// TwinCAT 3 PLC project TwinCAT_NC_Sample_Flying_Saw
// libraries:
//   Tc2_Math, * (Beckhoff Automation GmbH)
//   Tc2_MC2, * (Beckhoff Automation GmbH)
//   Tc2_MC2_FlyingSaw, * (Beckhoff Automation GmbH)
//   Tc2_Standard, * (Beckhoff Automation GmbH)
//   Tc2_System, * (Beckhoff Automation GmbH)
//   Tc3_Module, * (Beckhoff Automation GmbH)
// project tree:
//   Data types/ ST_AxisIn.TcDUT, ST_Axis.TcDUT, ST_AxisOut.TcDUT
//   Global Variables/ Globale_Variablen.TcGVL, GVL_FlyingSaw.TcGVL
//   / GlobalTextList.TcGTLO, PlcTask.TcTTO, Visualization Manager.TcVMO (not stored), VISU_TASK.TcTTO
//   POUs/ FB_Motion.TcPOU, MAIN.TcPOU, PRG_FlyingSaw.TcPOU, PRG_Simulation.TcPOU
//   Visualizations/ ImagePool.TcIPO (not stored), TC_FlyingSawPage.TcVIS
// real-time tasks:
//   TASK PlcTask: cycle T#10ms, priority 20, ADS port 350
//   TASK VISU_TASK: cycle T#10ms, priority 30, ADS port 351
// motion (NC):
//   TASK NC-Task 1 SAF: cycle T#2ms, priority 4, ADS port 501
//   TASK NC-Task 1 SVB: cycle T#10ms, priority 8, ADS port 511
//   AXIS Axis 1 (id 1)
//     Velo: Maximum=8000
//     OtherSettings: AllowMotionCmdToSlave=true
//     encoder EncType=1
//       EncPara: ModuloFactor=20000
//     drive DrvType=5
//       Analog: VeloReferenz=8200, ScaleFactorActTorque=0.1
//       TimeComp: TaskDelayCycles=1
//     controller CtrType=1
//       CtrPara: PriorControlFactor=1
//         Observer: BandWidth=20
//   AXIS Axis 2 (id 2)
//     Velo: Maximum=8000
//     OtherSettings: AllowMotionCmdToSlave=true
//     encoder EncType=1
//     drive DrvType=5
//       Analog: VeloReferenz=8200, ScaleFactorActTorque=0.1
//       TimeComp: TaskDelayCycles=1
//     controller CtrType=1
//       CtrPara: PriorControlFactor=1
//         Observer: BandWidth=20
//   AXIS Axis 3 (id 3)
//     OtherSettings: AllowMotionCmdToSlave=true
//     encoder EncType=1
//     drive DrvType=5
//       Analog: ScaleFactorActTorque=0.1
//       TimeComp: TaskDelayCycles=1
//     controller CtrType=1
//       CtrPara: PriorControlFactor=1
//         Observer: BandWidth=20
// variable links:
//   TwinCAT_NC_Sample_Flying_Saw/TwinCAT_NC_Sample_Flying_Saw Instance <-> NC-Task 1 SAF/Axes/Axis 1
//     PlcTask Inputs/.Axis1.NcToPlc <-> Outputs/ToPlc
//     PlcTask Outputs/.Axis1.PlcToNc <-> Inputs/FromPlc
//   TwinCAT_NC_Sample_Flying_Saw/TwinCAT_NC_Sample_Flying_Saw Instance <-> NC-Task 1 SAF/Axes/Axis 2
//     PlcTask Inputs/.Axis2.NcToPlc <-> Outputs/ToPlc
//     PlcTask Outputs/.Axis2.PlcToNc <-> Inputs/FromPlc
//   TwinCAT_NC_Sample_Flying_Saw/TwinCAT_NC_Sample_Flying_Saw Instance <-> NC-Task 1 SAF/Axes/Axis 3
//     PlcTask Inputs/.Axis3.NcToPlc <-> Outputs/ToPlc
//     PlcTask Outputs/.Axis3.PlcToNc <-> Inputs/FromPlc

CONFIGURATION TwinCAT_NC_Sample_Flying_Saw
    RESOURCE PLC ON TwinCAT3
        TASK PlcTask(INTERVAL := T#10ms, PRIORITY := 20);
        TASK VISU_TASK(INTERVAL := T#10ms, PRIORITY := 30);
        PROGRAM MAIN WITH PlcTask : MAIN;
        PROGRAM VisuElems_Visu_Prg WITH VISU_TASK : VisuElems.Visu_Prg;
    END_RESOURCE
END_CONFIGURATION

// ---- Data types/ST_AxisIn.TcDUT
TYPE ST_AxisIn :
STRUCT
	bEnable				: BOOL;
	bMoveAbs			: BOOL;
	bManuelIleri		: BOOL;
	bManuelGeri			: BOOL;
	bReset				: BOOL;
	bStop				: BOOL;
	bMoveVelo			: BOOL;
	bGearInPos			: BOOL;
	bGearOut			: BOOL;
	bMcMoveModulo		: BOOL;
	bSetPosition		: BOOL;
	
	
	fPos				: LREAL;
	fVelo				: LREAL;
	fOverride			: LREAL;
	fMaxCoupleVelo		: LREAL;
	fMasterGearPos		: LREAL;
	fSlaveGearPos		: LREAL;
	fMasterStartDistance: LREAL;
	
END_STRUCT
END_TYPE

// ---- Data types/ST_Axis.TcDUT
TYPE ST_Axis :
STRUCT
	IN	: ST_AxisIn;
	OUT	: ST_AxisOut;
	
END_STRUCT
END_TYPE

// ---- Data types/ST_AxisOut.TcDUT
TYPE ST_AxisOut :
STRUCT
	bMoveAbsDone	: BOOL;
	bMoveAbsBusy	: BOOL;
	bMoveAbsErr		: BOOL;
	bResetDone		: BOOL;
	bStopDone		: BOOL;
	bEnabled		: BOOL;
	bMoveVeloDone	: BOOL;
	bMoveVeloBusy	: BOOL;
	bCoupled		: BOOL;
	bDecoupled		: BOOL;
	bCoupleErr		: BOOL;
	bMoveModuloDone	: BOOL;
	bMoveModuloBusy	: BOOL;
	bMoveModuloErr	: BOOL;
	bSetPositionDone: BOOL;
	
END_STRUCT
END_TYPE

// ---- Global Variables/Globale_Variablen.TcGVL
{attribute 'Tc2GvlVarNames'}
VAR_GLOBAL
	Axis1		: AXIS_REF;
	Axis2		: AXIS_REF;
	Axis3		: AXIS_REF;
	//Axis4		: AXIS_REF;
	
	stAxis1		: ST_Axis;
	stAxis2		: ST_Axis;
	stAxis3		: ST_Axis;

	fbMotion1	: FB_Motion;
	fbMotion2	: FB_Motion;
	fbMotion3	: FB_Motion;
	
	
	bEnable		: BOOL;

END_VAR

// ---- Global Variables/GVL_FlyingSaw.TcGVL
VAR_GLOBAL
	bStartSensor: BOOL;
	bProcessActive: BOOL;
	nLastState: INT;
	bAsagi: BOOL;
	bYukari: BOOL;
	bYukariSensor: BOOL;
	bBaslat: BOOL;
	bMalzemeSensoru: BOOL;
	i: DINT;
	rProcessActive: R_TRIG;
	fCalculate: LREAL;
	fbMcSetPosition: MC_SetPosition;
END_VAR

// ---- POUs/MAIN.TcPOU
PROGRAM MAIN
(* 	Flying Saw synchronization of master and slave axes.
 *	The tool axis operates while master and slave are synchronized
 *	The operation takes place consequently after a constant distance 
 *	of the master. This is a typical cutting precedure.
 *)
VAR 
	
	

END_VAR

fbMotion1(Axis:= Axis1, stAxis:= stAxis1 , Slave:= Axis2);
fbMotion2(Axis:= Axis2,stAxis:= stAxis2 , Slave:= Axis1);
fbMotion3(Axis:= Axis3,stAxis:= stAxis3 , Slave:= Axis2);

IF bEnable THEN
	stAxis1.IN.bEnable		:= TRUE;
	stAxis1.IN.fOverride	:= 100;
	stAxis2.IN.bEnable		:= TRUE;
	stAxis2.IN.fOverride	:= 100;
	stAxis3.IN.bEnable		:= TRUE;
	stAxis3.IN.fOverride	:= 100;
ELSE
	stAxis1.IN.bEnable		:= FALSE;
	stAxis1.IN.fOverride	:= 0;
	stAxis2.IN.bEnable		:= FALSE;
	stAxis2.IN.fOverride	:= 0;
	stAxis3.IN.bEnable		:= FALSE;
	stAxis3.IN.fOverride	:= 0;
END_IF

PRG_FlyingSaw();
PRG_Simulation();

END_PROGRAM

// ---- POUs/PRG_FlyingSaw.TcPOU
PROGRAM PRG_FlyingSaw
VAR
	nState: INT;

	sMsg: STRING(INT#30);
END_VAR

rProcessActive(CLK:= bProcessActive , Q=> );
IF rProcessActive.Q THEN
			i	:= i+1;
END_IF

CASE nState OF
	
0:
	IF bStartSensor THEN
		nState	:= 5;
		bProcessActive	:= TRUE;
	END_IF

5:
	IF stAxis1.OUT.bEnabled AND stAxis2.OUT.bEnabled AND stAxis3.OUT.bEnabled THEN
		nState	:= 10;	
	END_IF
	
10:	
	stAxis1.IN.bMoveAbs		:= TRUE;
	stAxis1.IN.fVelo				:= 3000;
	stAxis1.IN.fPos					:= 20000;
	IF stAxis1.OUT.bMoveAbsBusy AND NOT stAxis1.OUT.bMoveAbsErr THEN
		nState						:= 20;
		//stAxis1.IN.bMcMoveModulo	:= FALSE;
	ELSIF stAxis1.OUT.bMoveAbsErr THEN
		nLastState					:= nState;		
		stAxis1.IN.bMcMoveModulo	:= FALSE;
		nState						:= 999;
	END_IF
	
20:
	fCalculate	:= (((DINT_TO_LREAL(i-1))*20000)+1000);
	IF Axis1.NcToPlc.ModuloActPos >= 1000 THEN
		nState	:= 30;
	ELSIF axis1.Status.Error THEN
		nState	:= 999;
	END_IF
	
30:
	stAxis1.IN.bGearInPos			:= TRUE;
	stAxis1.IN.fMasterGearPos		:= 6000;
	stAxis1.IN.fSlaveGearPos		:= 1000;

	(*
	IF i=1 THEN
		stAxis1.IN.fMasterGearPos		:= 6000;
		stAxis1.IN.fSlaveGearPos		:= 1000;
		stAxis1.IN.fMasterStartDistance	:= 0;
	ELSE
		stAxis1.IN.fMasterGearPos		:= 6000+(20000*DINT_TO_LREAL(i));
		stAxis1.IN.fSlaveGearPos		:= 1000;
		stAxis1.IN.fMasterStartDistance	:= 20000*i;
	END_IF*)
	IF stAxis1.OUT.bCoupled AND NOT stAxis1.OUT.bCoupleErr THEN
		nState					:= 40;
		stAxis1.IN.bGearInPos	:= FALSE;
		sMsg					:= 'Flying Saw Hareketi Basladi...';
	ELSIF stAxis1.OUT.bCoupleErr THEN
	//	stAxis1.IN.bGearInPos	:= FALSE;
		nState					:= 999;
	END_IF
	
40:	
	IF Axis2.NcToPlc.ActPos>=1000 THEN
		nState		:= 50;
	ELSIF axis2.Status.Error THEN
		nState		:= 999;
	END_IF
		
50:
	stAxis3.IN.bMoveAbs				:= TRUE;
	stAxis3.IN.fVelo				:= 2000;
	stAxis3.IN.fPos					:= 1000;
	IF stAxis3.OUT.bMoveAbsBusy AND NOT stAxis3.OUT.bMoveAbsErr THEN
		nState				:= 60;
		stAxis3.IN.bMoveAbs	:= FALSE;
	ELSIF stAxis3.OUT.bMoveAbsErr THEN
		nState				:= 999;
		stAxis3.IN.bMoveAbs	:= FALSE;
	END_IF

60:
	IF stAxis3.OUT.bMoveAbsDone  AND NOT stAxis3.OUT.bMoveAbsErr  THEN
		nState				:= 70;
	ELSIF stAxis3.OUT.bMoveAbsErr  THEN
		nState				:= 999;
	END_IF
	
70:
	stAxis3.IN.bMoveAbs		:= TRUE;
	stAxis3.IN.fVelo		:= 1000;
	stAxis3.IN.fPos			:= 0;
	IF stAxis3.OUT.bMoveAbsBusy AND NOT stAxis3.OUT.bMoveAbsErr THEN
		nState				:= 80;
		stAxis3.IN.bMoveAbs	:= FALSE;
	ELSIF stAxis3.OUT.bMoveAbsErr THEN
		nState				:= 999;
		stAxis3.IN.bMoveAbs	:= FALSE;
	END_IF
	
80:
	IF stAxis3.OUT.bMoveAbsDone  AND NOT stAxis3.OUT.bMoveAbsErr  THEN
		nState				:= 90;
	ELSIF stAxis3.OUT.bMoveAbsErr  THEN
		nState				:= 999;
	END_IF
	
90:
	stAxis1.IN.bGearOut := TRUE;
	IF stAxis1.OUT.bDecoupled THEN
		stAxis1.IN.bGearOut := FALSE;
		nState				:= 100;
		sMsg				:= 'Flying Saw Hareketi Sonlandi...';
	END_IF
	
100:
	stAxis2.IN.bStop	:= TRUE;
	IF stAxis2.OUT.bStopDone THEN
		nState			:= 110;
		stAxis2.IN.bStop:= FALSE;
	END_IF
	
110:
	stAxis2.IN.bMoveAbs	:= TRUE;
	stAxis2.IN.fVelo	:= 7000;
	stAxis2.IN.fPos		:= 0;
	IF stAxis2.OUT.bMoveAbsBusy AND NOT stAxis2.OUT.bMoveAbsErr  THEN
		nState	:= 120;
	//	stAxis2.IN.bMoveAbs	:= FALSE;	
	ELSIF stAxis2.OUT.bMoveAbsErr  THEN
		nState	:= 99;		
		stAxis2.IN.bMoveAbs	:= FALSE;	
	END_IF
	
120:
	IF stAxis2.OUT.bMoveAbsDone AND NOT stAxis2.OUT.bMoveAbsErr  THEN
		nState	:= 130;
	ELSIF stAxis2.OUT.bMoveAbsErr  THEN
		nState		:= 99;
	END_IF
	

(*	
140:
	stAxis1.IN.bMcMoveModulo		:= TRUE;
	stAxis1.IN.fVelo				:= 2000;
	stAxis1.IN.fPos					:= 0;
	IF stAxis1.OUT.bMoveModuloBusy AND NOT stAxis1.OUT.bMoveModuloErr THEN
		nState						:= 150;
		stAxis1.IN.bMcMoveModulo	:= FALSE;
	ELSIF stAxis1.OUT.bMoveModuloErr THEN
		nLastState					:= nState;		
		stAxis1.IN.bMcMoveModulo	:= FALSE;
		nState						:= 999;
	END_IF
	
150:
	IF stAxis1.OUT.bMoveModuloDone THEN
		nState			:= 160;
		bProcessActive	:= FALSE;
	ELSIF stAxis1.OUT.bMoveModuloErr THEN
		nState			:= 999;
	END_IF
	*)
160:
	stAxis1.IN.bSetPosition		:= TRUE;
	IF stAxis1.OUT.bSetPositionDone THEN
		stAxis1.IN.bSetPosition	:= FALSE;
		nState					:= 0;
		bProcessActive			:= FALSE;
	END_IF
	
999:
;

END_CASE

IF stAxis1.OUT.bMoveAbsDone AND stAxis2.OUT.bMoveAbsDone  THEN
	nState	:= 160;
	stAxis1.IN.bMoveAbs	:= FALSE;		
	stAxis2.IN.bMoveAbs	:= FALSE;	
ELSIF stAxis1.OUT.bMoveAbsErr THEN
	nState	:= 999;
	stAxis1.IN.bMoveAbs	:= FALSE;	
END_IF


IF NOT bProcessActive AND NOT bStartSensor AND bMalzemeSensoru THEN
		bAsagi		:= TRUE;
		bYukari		:= FALSE;
ELSIF bStartSensor THEN
		bAsagi		:= FALSE;
		bYukari		:= TRUE;
ELSIF bYukariSensor THEN
		bYukari		:= FALSE;
		bAsagi		:= FALSE;
END_IF

END_PROGRAM

// ---- POUs/PRG_Simulation.TcPOU
PROGRAM PRG_Simulation
VAR
	fAxis3SimulationActPosY: LREAL;
	bParca1Invisible: BOOL;
	bParca2Invisible2: BOOL;
	fAxis1SimulationActPosX: LREAL;

	fAxis2SimulationActPosX: LREAL;
	bMatkapInvisible: BOOL;
	bMatkapInvisible2: BOOL;
	bMatkapInvisible3: BOOL;
	nState: INT;
	nUp: INT;
	bParcaUpInvisible: BOOL;
	nRight: INT;
	bParcaRightInvisible: BOOL;
	t1: TON;
	bAxis31000Position: BOOL;
END_VAR

IF Axis1.NcToPlc.ActPos >= 6000 AND Axis1.NcToPlc.ActPos < 20000 THEN
	bParca1Invisible		:= TRUE;
	bParca2Invisible2		:= FALSE;
	fAxis1SimulationActPosX	:= (Axis1.NcToPlc.ActPos-6000)/30;
ELSIF Axis1.NcToPlc.ActPos >= 20000 THEN
	bParca2Invisible2		:= TRUE;
	bAxis31000Position		:= FALSE;
	fAxis3SimulationActPosY	:= 0;
ELSIF Axis1.NcToPlc.ActPos=0 OR Axis1.NcToPlc.ActPos<1 THEN
	bParca2Invisible2		:= TRUE;
END_IF

IF Axis2.NcToPlc.ActPos>=1000 AND Axis2.Status.PositiveDirection THEN
	fAxis2SimulationActPosX	:= (Axis2.NcToPlc.ActPos-1000)/30;
	bMatkapInvisible		:= TRUE;
	bMatkapInvisible2		:= FALSE;
ELSIF Axis2.NcToPlc.ActPos=0 OR Axis2.NcToPlc.ActPos<1 THEN
	bMatkapInvisible		:= FALSE;
	bMatkapInvisible3		:= TRUE;
	bMatkapInvisible2		:= TRUE;
END_IF


IF Axis2.Status.NegativeDirection THEN
	fAxis2SimulationActPosX	:= (Axis2.NcToPlc.ActPos)/30;
	bMatkapInvisible	:= TRUE;
	bMatkapInvisible2	:= TRUE;
	bMatkapInvisible3	:= FALSE;
END_IF

IF Axis3.NcToPlc.ActPos>=692.3076921 AND NOT bAxis31000Position THEN
	fAxis3SimulationActPosY	:= (Axis3.NcToPlc.ActPos/15.38461538)-45;
END_IF

IF  Axis3.NcToPlc.ActPos>=999 THEN
	fAxis3SimulationActPosY	:= 20;
	bAxis31000Position		:= TRUE;
END_IF

CASE nState OF

0:
	.bStartSensor	:= FALSE;
	IF NOT .bProcessActive THEN
		.bEnable	:= TRUE;
		nState		:= 10;
		bParcaUpInvisible	:= FALSE; 
	END_IF

10:
	nUp						:= nUp+1;
	IF nUp>=135 THEN
		nState				:= 20;
	END_IF
	
20:
	nRight					:= nRight+1;
	IF nRight>=61 THEN
		bParcaUpInvisible	:= TRUE; 
		nState				:= 25;
		bParca1Invisible		:= FALSE;
	END_IF
	
25:
	nRight					:= nRight-1;
	IF nRight<=0 THEN		
		nState				:= 27;	
	END_IF

27:
	nUp						:= nUp-1;
	IF nUp<=0 THEN
		nState				:= 30;
	END_IF
30:
	bStartSensor				:= TRUE;
	t1(IN:= TRUE , PT:= T#30MS , Q=> , ET=> );
	IF t1.Q THEN
		t1(IN:= FALSE);
		nState						:= 0;
		nRight						:= 0;
		nUp							:= 0;
	END_IF

END_CASE

END_PROGRAM

// ---- POUs/FB_Motion.TcPOU
FUNCTION_BLOCK FB_Motion
VAR_INPUT
	
END_VAR
VAR_OUTPUT

END_VAR
VAR
	fbMcPower	: MC_Power;
	fbMcJog		: MC_Jog;
	fbMcReset: MC_Reset;
	fbMcStop: MC_Stop;
	fbMcMoveAbs: MC_MoveAbsolute;
	fbMcGearInPos: MC_GearInPos;
	fbMcMoveModulo: MC_MoveModulo;
	fbMcGearOut: MC_GearOut;
	fbMcReadStatus: MC_ReadStatus;
	fbMcSetPosition: MC_SetPosition;
END_VAR
VAR_IN_OUT
	stAxis	: ST_Axis;
	Axis	: AXIS_REF;
	Slave	: AXIS_REF;
END_VAR

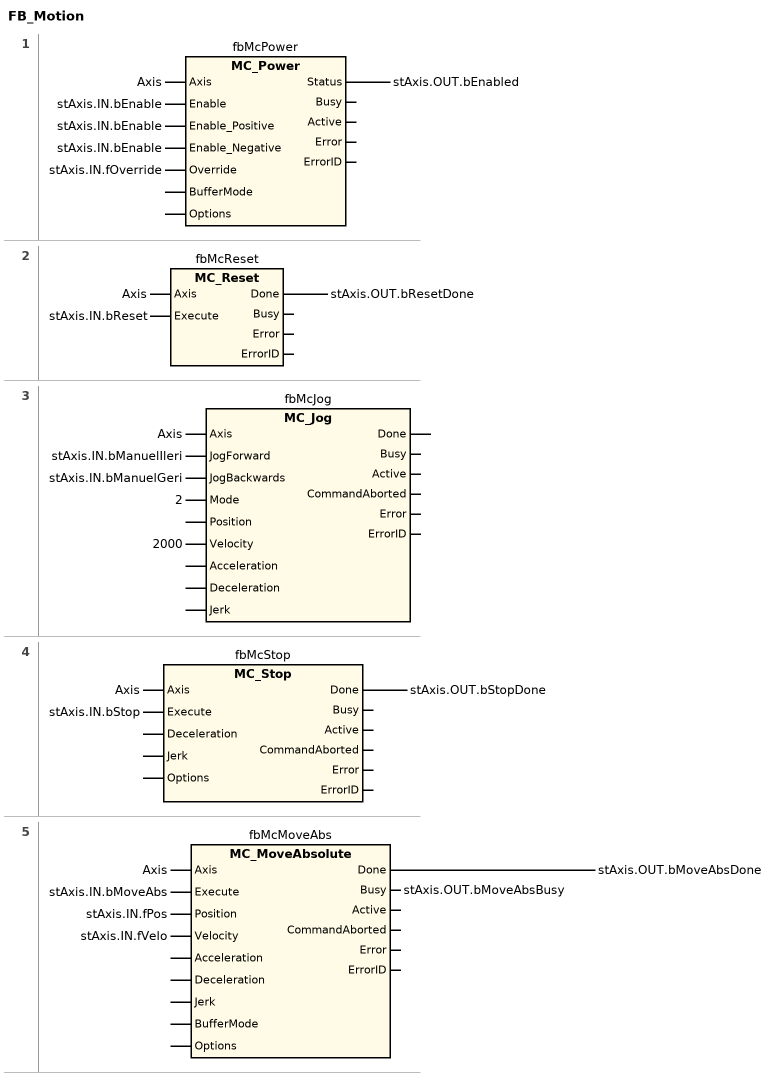
// NETWORK 1
fbMcPower(
    Axis := Axis,
    Enable := stAxis.IN.bEnable,
    Enable_Positive := stAxis.IN.bEnable,
    Enable_Negative := stAxis.IN.bEnable,
    Override := stAxis.IN.fOverride); // MC_Power
stAxis.OUT.bEnabled := fbMcPower.Status;

// NETWORK 2
fbMcReset(Axis := Axis, Execute := stAxis.IN.bReset); // MC_Reset
stAxis.OUT.bResetDone := fbMcReset.Done;

// NETWORK 3
fbMcJog(
    Axis := Axis,
    JogForward := stAxis.IN.bManuelIleri,
    JogBackwards := stAxis.IN.bManuelGeri,
    Mode := 2,
    Velocity := 2000); // MC_Jog

// NETWORK 4
fbMcStop(Axis := Axis, Execute := stAxis.IN.bStop); // MC_Stop
stAxis.OUT.bStopDone := fbMcStop.Done;

// NETWORK 5
fbMcMoveAbs(
    Axis := Axis,
    Execute := stAxis.IN.bMoveAbs,
    Position := stAxis.IN.fPos,
    Velocity := stAxis.IN.fVelo,
    Busy => stAxis.OUT.bMoveAbsBusy); // MC_MoveAbsolute
stAxis.OUT.bMoveAbsDone := fbMcMoveAbs.Done;

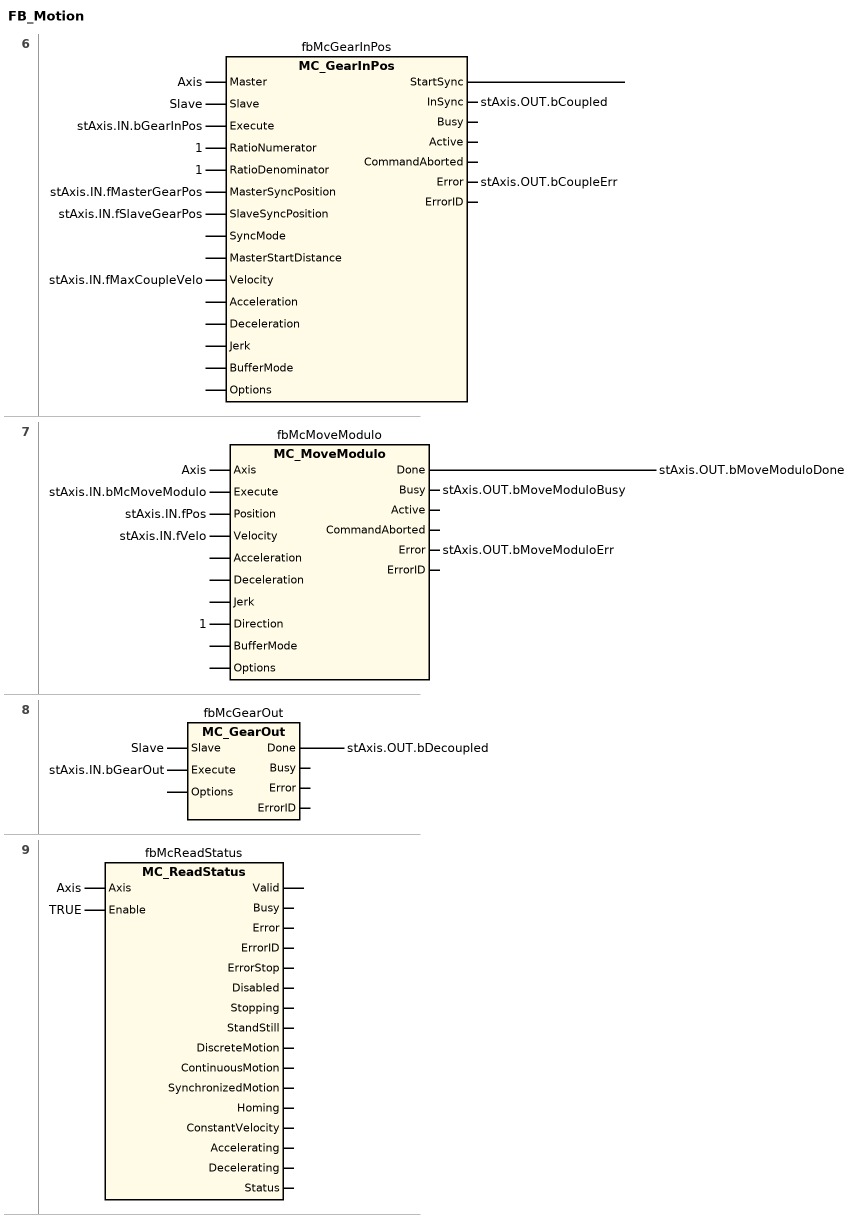
// NETWORK 6
fbMcGearInPos(
    Master := Axis,
    Slave := Slave,
    Execute := stAxis.IN.bGearInPos,
    RatioNumerator := 1,
    RatioDenominator := 1,
    MasterSyncPosition := stAxis.IN.fMasterGearPos,
    SlaveSyncPosition := stAxis.IN.fSlaveGearPos,
    Velocity := stAxis.IN.fMaxCoupleVelo,
    InSync => stAxis.OUT.bCoupled,
    Error => stAxis.OUT.bCoupleErr); // MC_GearInPos

// NETWORK 7
fbMcMoveModulo(
    Axis := Axis,
    Execute := stAxis.IN.bMcMoveModulo,
    Position := stAxis.IN.fPos,
    Velocity := stAxis.IN.fVelo,
    Direction := 1,
    Busy => stAxis.OUT.bMoveModuloBusy,
    Error => stAxis.OUT.bMoveModuloErr); // MC_MoveModulo
stAxis.OUT.bMoveModuloDone := fbMcMoveModulo.Done;

// NETWORK 8
fbMcGearOut(Slave := Slave, Execute := stAxis.IN.bGearOut); // MC_GearOut
stAxis.OUT.bDecoupled := fbMcGearOut.Done;

// NETWORK 9
fbMcReadStatus(Axis := Axis, Enable := TRUE); // MC_ReadStatus

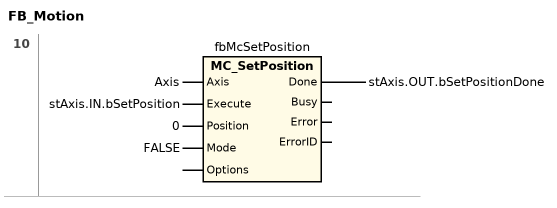
// NETWORK 10
fbMcSetPosition(Axis := Axis, Execute := stAxis.IN.bSetPosition, Position := 0, Mode := FALSE); // MC_SetPosition
stAxis.OUT.bSetPositionDone := fbMcSetPosition.Done;

END_FUNCTION_BLOCK

// ---- GlobalTextList.TcGTLO
TEXTLIST GlobalTextList
  646 = '%s'
  892 = 'ENABLE'
  111 = 'START'
END_TEXTLIST

// ---- Visualizations/TC_FlyingSawPage.TcVIS
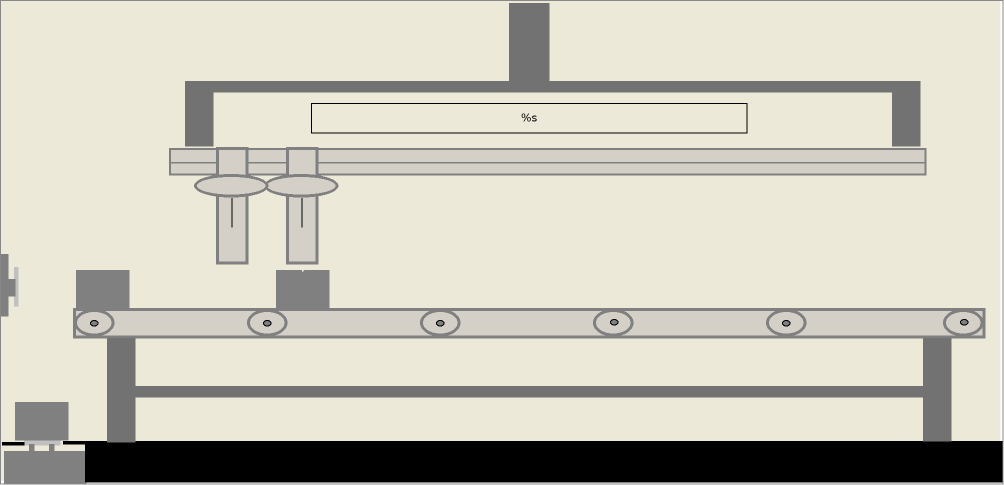
VISUALIZATION TC_FlyingSawPage  // 1004x485
    Rectangle (0,0 1000x480)
    RoundedRectangle (169,148 757x27)
    Rectangle (171,162 755x1)
    RoundedRectangle (73,308 912x30)
    Rectangle (4,451 82x32)
    RoundedRectangle (24,440 36x5)
        p2738717112: -(PRG_Simulation.nUp)
    Rectangle (85,441 917x41)
    Rectangle (63,441 34x3)
    Rectangle (29,444 5x8)
        p2773130477: -(PRG_Simulation.nUp)
    RoundedRectangle (49,444 5x8)
        p2773130477: -(PRG_Simulation.nUp)
    Rectangle (216,147 32x117), invisible if: PRG_Simulation.bMatkapInvisible
        p3560616238: Axis2.NcToPlc.ActPos/14.706
    Ellipse (194,174 74x23), invisible if: PRG_Simulation.bMatkapInvisible
        p2738717112: (Axis3.NcToPlc.ActPos)/15.38461538
        p3560616238: Axis2.NcToPlc.ActPos/14.706
    Line (232,227) (232,198), invisible if: PRG_Simulation.bMatkapInvisible
        p2738717112: (Axis3.NcToPlc.ActPos)/15.38461538
        p3560616238: Axis2.NcToPlc.ActPos/14.706
    Rectangle (76,270 53x38), invisible if: PRG_Simulation.bParca1Invisible
        p3560616238: Axis1.NcToPlc.ActPos/30
    Rectangle (276,270 53x38), invisible if: PRG_Simulation.bParca2Invisible2
        p3560616238: PRG_Simulation.fAxis1SimulationActPosX
    Rectangle (286,147 32x117), invisible if: PRG_Simulation.bMatkapInvisible2
        p3560616238: PRG_Simulation.fAxis2SimulationActPosX
    Ellipse (264,174 74x23), invisible if: PRG_Simulation.bMatkapInvisible2
        p2738717112: (Axis3.NcToPlc.ActPos)/15.38461538
        p3560616238: PRG_Simulation.fAxis2SimulationActPosX
    Rectangle (216,147 32x117), invisible if: PRG_Simulation.bMatkapInvisible3
        p3560616238: PRG_Simulation.fAxis2SimulationActPosX
    Ellipse (194,174 74x23), invisible if: PRG_Simulation.bMatkapInvisible3
        p2738717112: (Axis3.NcToPlc.ActPos)/15.38461538
        p3560616238: PRG_Simulation.fAxis2SimulationActPosX
    Line (232,227) (232,198), invisible if: PRG_Simulation.bMatkapInvisible3
        p2738717112: (Axis3.NcToPlc.ActPos)/15.38461538
        p3560616238: PRG_Simulation.fAxis2SimulationActPosX
    Rectangle (15,402 53x38), invisible if: PRG_Simulation.bParcaUpInvisible
        p3560616238: PRG_Simulation.nRight
        p2738717112: -(PRG_Simulation.nUp)
    Rectangle (2,442 22x3)
    Rectangle (0,254 8x62)
    Rectangle (14,267 4x39)
        p3560616238: PRG_Simulation.nRight
    Rectangle (8,279 7x17)
        p874137650: PRG_Simulation.nRight
    Rectangle (302,270 1x1), invisible if: PRG_Simulation.bParca2Invisible2
        p3560616238: PRG_Simulation.fAxis2SimulationActPosX
        p2773130477: PRG_Simulation.fAxis3SimulationActPosY
    Line (302,227) (302,198), invisible if: PRG_Simulation.bMatkapInvisible2
        p2738717112: (Axis3.NcToPlc.ActPos)/15.38461538
        p3560616238: PRG_Simulation.fAxis2SimulationActPosX
    Ellipse (74,309 40x27)
    Ellipse (247,309 40x27)
    Ellipse (420,309 40x27)
    Ellipse (593,309 40x27)
    Ellipse (766,309 40x27)
    Ellipse (943,309 40x27)
    Ellipse (90,320 8x6)
    Ellipse (263,320 8x6)
    Ellipse (436,320 8x6)
    Ellipse (610,319 8x6)
    Ellipse (782,320 8x6)
    Ellipse (960,319 8x6)
    Rectangle (107,338 28x104)
    Rectangle (923,338 28x103)
    Rectangle (131,386 794x11)
    Rectangle (185,81 735x11)
    Rectangle (892,90 28x56)
    Rectangle (185,90 28x56)
    Rectangle (509,3 40x79)
    Rectangle (311,103 436x30), "%s", text variable: PRG_FlyingSaw.sMsg
END_VISUALIZATION
